// TIA Portal V17 export
// export: Created 2022-07-20T06:59:47.7070424Z, ExportSetting WithDefaults, DisplayName Totally Integrated Automation Portal, DisplayVersion V17, DisplayName TIA Portal Openness, DisplayVersion V17, DisplayName TIA Portal Version Control Interface, DisplayVersion V17, DisplayName SINAMICS Startdrive Advanced, DisplayVersion V17, DisplayName SINAMICS Startdrive G130, G150, S120, S150, SINAMICS MV, S210, DisplayVersion V17, DisplayName SINAMICS Startdrive G110M, G120, G120C, G120D, G120P, G115D, DisplayVersion V17, DisplayName STEP 7 Professional, DisplayVersion V17, DisplayName STEP 7 Safety, DisplayVersion V17, DisplayName WinCC Advanced, DisplayVersion V17
FUNCTION_BLOCK "FB10160_FlexoInkCircuit"   // FB10160, LAD
TITLE = FB10160_FlexoInkCircuit
{ S7_Optimized_Access := 'TRUE' }
AUTHOR : Anirouddh
FAMILY : 1016x_FLEXO
VERSION : 1.0
// Release note : 
// 1.0 - Feature developped
// stored: AutoNumber false, IsIECCheckEnabled false, IsRetainMemResEnabled false, MemoryReserve 100, SetENOAutomatically false, UDAEnableTagReadback false
   VAR_INPUT
      ActivateRegulation : Bool;
      VarnishSensor : Bool;
      OperatorPadSensor : Bool;
      OppositePadSensor : Bool;
      RequestVarnishPumpActivation : Bool;
      RequestWashupPumpActivation : Bool;
      VerticalRollerInOriginPosition : Bool;
   END_VAR
   VAR_OUTPUT
      ActiveVarnishPump : Bool;
      ActiveWashupPump : Bool;
   END_VAR
   VAR
      R_TRIG_RequestVarnishPumpActivation : R_TRIG;
      R_TRIG_RequestWashupPumpActivation { S7_SetPoint := 'True'} : R_TRIG;
   END_VAR
BEGIN

REGION Network 1 (SCL): Edge Signals Management
   #R_TRIG_RequestVarnishPumpActivation(CLK:= #OperatorPadSensor AND #OppositePadSensor AND #RequestVarnishPumpActivation);
   #R_TRIG_RequestWashupPumpActivation(CLK := #VerticalRollerInOriginPosition AND #RequestWashupPumpActivation);
END_REGION

REGION Network 2 (SCL): Varnish Pump Management
   IF #ActivateRegulation THEN
       IF #VarnishSensor THEN
           #ActiveVarnishPump := FALSE;
       ELSE
           #ActiveVarnishPump := TRUE;
       END_IF;
   ELSE
       IF #R_TRIG_RequestVarnishPumpActivation.Q THEN
           #ActiveVarnishPump := TRUE;
       ELSIF NOT (#RequestVarnishPumpActivation) THEN
           #ActiveVarnishPump := FALSE;
       END_IF;
   END_IF;
END_REGION

REGION Network 3 (SCL): Washup Pump Management
   IF #VerticalRollerInOriginPosition AND #RequestWashupPumpActivation THEN
       #ActiveWashupPump := TRUE;
   ELSE
       #ActiveWashupPump := FALSE;
   END_IF;
END_REGION
END_FUNCTION_BLOCK
